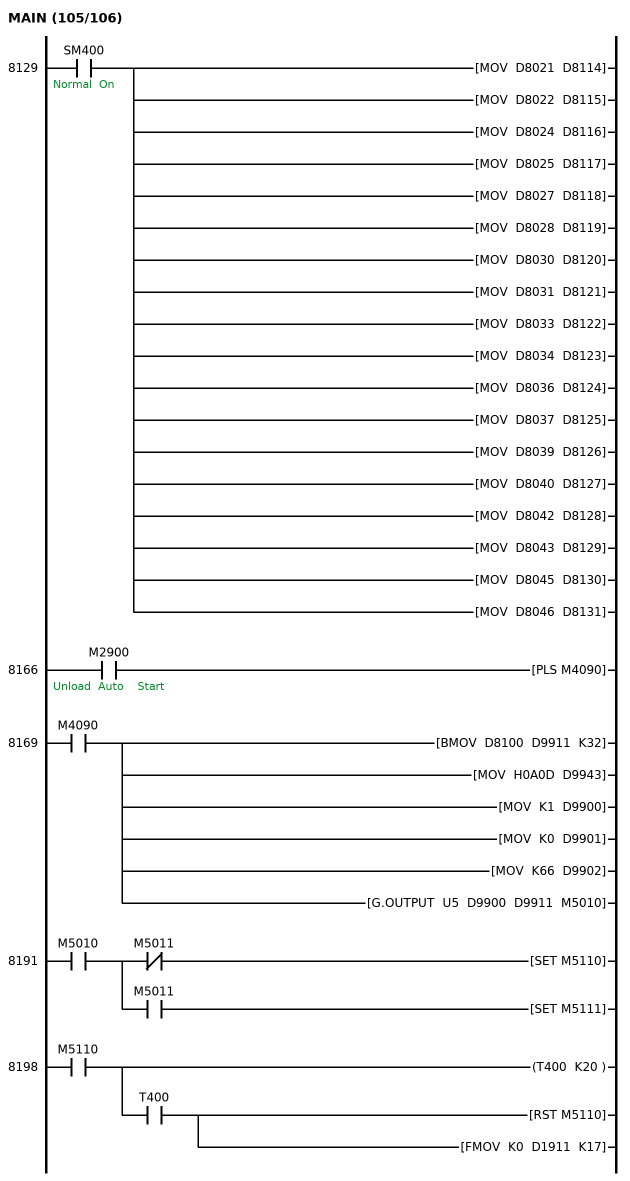
[picture p384: ladder of MAIN, rungs at steps 8129 to 8198]
8129  LD      SM400  ; Normal  On
      MOV     D8021 D8114
      MOV     D8022 D8115
      MOV     D8024 D8116
      MOV     D8025 D8117
      MOV     D8027 D8118
      MOV     D8028 D8119
      MOV     D8030 D8120
      MOV     D8031 D8121
      MOV     D8033 D8122
      MOV     D8034 D8123
      MOV     D8036 D8124
      MOV     D8037 D8125
      MOV     D8039 D8126
      MOV     D8040 D8127
      MOV     D8042 D8128
      MOV     D8043 D8129
      MOV     D8045 D8130
      MOV     D8046 D8131
8166  LD      M2900  ; Unload  Auto    Start
      PLS     M4090
8169  LD      M4090
      BMOV    D8100 D9911 K32
      MOV     H0A0D D9943
      MOV     K1 D9900
      MOV     K0 D9901
      MOV     K66 D9902
      G.OUTPUT U5 D9900 D9911 M5010
8191  LD      M5010
      MPS
      ANI     M5011
      SET     M5110
      MPP
      AND     M5011
      SET     M5111
8198  LD      M5110
      OUT     T400 K20
      AND     T400
      RST     M5110
      FMOV    K0 D1911 K17
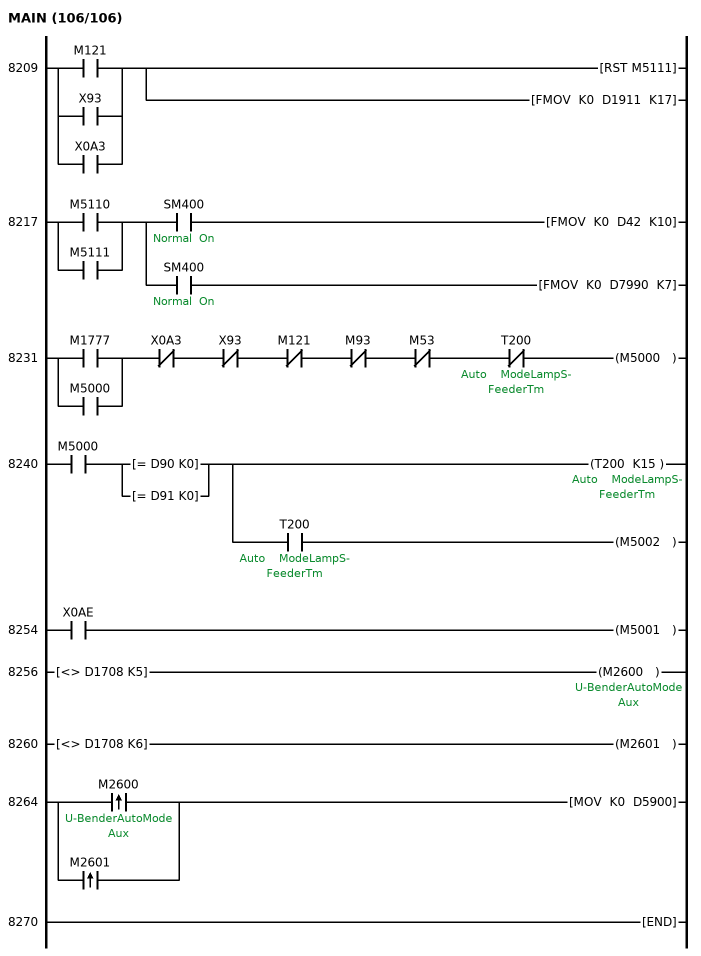
8209  LD      M121
      OR      X93
      OR      X0A3
      RST     M5111
      FMOV    K0 D1911 K17
8217  LD      M5110
      OR      M5111
      MPS
      AND     SM400  ; Normal  On
      FMOV    K0 D42 K10
      MPP
      AND     SM400  ; Normal  On
      FMOV    K0 D7990 K7
8231  LD      M1777
      OR      M5000
      ANI     X0A3
      ANI     X93
      ANI     M121
      ANI     M93
      ANI     M53
      ANI     T200  ; Auto    ModeLampS-FeederTm
      OUT     M5000
8240  LD      M5000
      LD=     D90 K0
      OR=     D91 K0
      ANB
      OUT     T200 K15  ; Auto    ModeLampS-FeederTm
      AND     T200  ; Auto    ModeLampS-FeederTm
      OUT     M5002
8254  LD      X0AE
      OUT     M5001
8256  LD<>    D1708 K5
      OUT     M2600  ; U-BenderAutoModeAux
8260  LD<>    D1708 K6
      OUT     M2601
8264  LDP     M2600  ; U-BenderAutoModeAux
      ORP     M2601
      MOV     K0 D5900
8270  END
END_PROGRAM

// device comments not shown above
D2  ; 150Ton  AutoBuff
R600  ; +OT Set PositionAxis-01
X31  ; f
X4B  ; Reset   #3
X4D  ; Reset   #2
X55  ; Carriage"B" OL
X56  ; Carriage"C" OL
X57  ; Carriage"D" OL
X58  ; Carriage"E" OL
X59  ; Carriage"F" OL
X80  ; NotchingSafety  Det'
X25D  ; NotchingR-SafetyDet'
X26B  ; NotchingR-Screp C/V OL
X303  ; 150Ton  BackPushUp Px
X304  ; 150Ton  BackPushDown Px
X305  ; 150Ton  SidePush1W-DetPx
X306  ; 150Ton  SidePush1RevPx
X30B  ; 150Ton  Safety#1Ls
X30C  ; 150Ton  Press UpPx
X30D  ; 150Ton  PressMidDet'Px
X30E  ; 150Ton  Press DnPx
X30F  ; 150Ton  PressureCheck
X313  ; 150Ton  Stopp UpPx
X314  ; 150Ton  Stopp DnPx
X315  ; 150Ton  SidePush2W-DetPx
X316  ; 150Ton  SidePush2Rev Px
X319  ; NotchingOil TempHigh
X31A  ; NotchingHi Press
X31B  ; 150Ton  Safety#1Ls
X31C  ; 150Ton  Side    L-Safety
X31D  ; 150Ton  Side    R-Safety
X31E  ; 150Ton  Hyd'TankTempHigh
X31F  ; 150Ton  Hyd'TankTempLow
X487  ; Buffer  Work    Stop
X490  ; Divert#2WorkDet'#1
X49E  ; Z-BenderHyd' OilTemp Hi
X54C  ; L-BendOtSideMoldPOt Fwd
X54D  ; L-BendOtSideMoldPOt Rev
X5CC  ; U-BendOtSideMoldPin Fwd
X5CD  ; U-BendOtSideMoldPin Rev
X5CE  ; U-BendOtUp GuideFwd
X600  ; U-BendInConv' Up
X601  ; U-BendInConv' Dn
X660  ; U-BendOtConv' Up
X661  ; U-BendOtConv' Dn
X6C0  ; Unload  Transfer+ OT
X6C1  ; Unload  TransferHome
X6C2  ; Unload  Transfer- OT
X6C8  ; Unload  TransferUp
X6C9  ; Unload  TransferDown
X6CA  ; Unload  Head    Clamp Px
X6CB  ; Unload  Head    Unclamp Px
X720  ; NEW SHEARING DIV. DN
X762  ; Buffer  Conv' OL
Y0B9  ; Buffer  Conv'Mc
Y0E4  ; Cycle Time Hold
Y0E5  ; Cycle Time Reset
Y1B6  ; Lifter  Up/Down Slow
Y1B7  ; Lifter  Up/Down Reset
Y2AA  ; NotchingRellief Sv
Y320  ; 150Ton  BackPushUp Sv
Y321  ; 150Ton  BackPushDn Sv
Y324  ; 150Ton  SidePushFwd Sv
Y325  ; 150Ton  SidePushRev Sv
Y326  ; NotchingHi PressSv
Y328  ; 150Ton  Stopper Up Sv
Y329  ; 150Ton  Stopper Dn Sv
Y32B  ; 150Ton  Press UpSv
Y32C  ; 150Ton  Press DnSv
Y32D  ; 150Ton  Rellief Sv
Y32E  ; 150Ton  Exhaust Sv
Y32F  ; 150Ton  WheelingSv
Y414  ; L-BenderRellief Sv
Y4AB  ; Z-BednerUp Sv
Y634  ; U-BendInSideGuidFwd Sv
Y694  ; U-BendOtSideGuidFwd Sv
Y6E0  ; Unload  TransferUp Sv
Y6E1  ; Unload  TransferDn Sv
Y74D  ; OutConv'#44MotorMc
Y74E  ; OutConv'#45MotorMc
Y79C  ; m43 cv lift up sol
M243  ; Divert#2On At
M248  ; Taping#1Work    Finish  Set
M278  ; IdleConvWork    Finish  Set
M282  ; IdleConvOn At
M283  ; U-BenderServo GoAt
M284  ; U-BenderOn At
M285  ; U-BenderOff At
M1001  ; Carriage"A" Set Sw
M1002  ; Carriage"B" Set Sw
M1003  ; Carriage"C" Set Sw
M1004  ; Carriage"D" Set Sw
M1005  ; Carriage"E" Set Sw
M1014  ; Sheet   Feeder  "E" Pos'Set Sw
M1015  ; Sheet   Feeder  "F" Pos'Set Sw
M1016  ; Sheet   Feeder  ConvPos'Set Sw
M1020  ; Sheet   Feeder  "A" Pos'Set Lp
M1021  ; Sheet   Feeder  "B" Pos'Set Lp
M1022  ; Sheet   Feeder  "C" Pos'Set Lp
M1023  ; Sheet   Feeder  "D" Pos'Set Lp
M1024  ; Sheet   Feeder  "E" Pos'Set Lp
M1025  ; Sheet   Feeder  "F" Pos'Set Lp
M1026  ; Sheet   Feeder  ConvPos'Set Lp
M1079  ; Carriage#2 Pos'  Fault
M1081  ; Carriage#4 Pos'  Fault
M1082  ; Carriage#5 Pos'  Fault
M1083  ; Carriage#6 Pos'  Fault
M1090  ; CarriagePositionOK
M1098  ; S/F     CarriageOK
M1102  ; S/F     Working Order Ok
M1118  ; S/F Car'PositionGo Aux.
M1230  ; 2-Axis  PositionOK
M1231  ; 3-Axis  PositionOK
M1232  ; 4-Axis  PositionOK
M1233  ; 5-Axis  PositionOK
M1234  ; 6-Axis  PositionOK
M1235  ; 7-Axis  PositionOK
M1236  ; 8-Axis  PositionOK
M1237  ; 2-Axis  PositionOK
M1238  ; 16-Axis PositionOK
M1316  ; NotchingMidStoppDown At
M1333  ; NotchingMid SidePush    Fwd At
M1401  ; 150Ton  Auto    Mode
M1402  ; 150Ton  Manual  Mode
M1410  ; 150Ton  Hold Sw
M1420  ; 150Ton  Press   Pass    Model
M1425  ; 150Ton  Working Model   Detect
M1430  ; 12-Axis PositionOK
M1431  ; 13-Axis PositionOK
M1439  ; 150Ton  All-AxisPos' OK
M1452  ; 150Ton  Press   Up Hm
M1453  ; 150Ton  BackPushRev Hm
M1454  ; 150Ton  BackPushDown Hm
M1455  ; 150Ton  Stopper Down Hm
M1456  ; 150Ton  SidePushRev Hm
M1471  ; 150Ton  Conv'RunEnable
M1472  ; 150Ton  ServoRunEnable
M1520  ; 150Ton  Press   Up Hm At
M1521  ; 150Ton  Stopper Up At
M1522  ; 150Ton  BackPushRev At
M1523  ; 150Ton  BackPushUp At
M1524  ; 150Ton  BackPushFwd At
M1525  ; 150Ton  SidePushFwd At
M1526  ; 150Ton  SidePush34Fwd At
M1528  ; 150Ton  Press   Down At
M1533  ; 150Ton  Press   Up At
M1534  ; 150Ton  SidePushBwd At
M1535  ; 150Ton  BackPushBwd At
M1536  ; 150Ton  SidePush#34BwdAt
M1537  ; 150Ton  BackPushDown At
M1538  ; 150Ton  Stopper Down At
M1560  ; 150Ton  Press   Stop
M1580  ; 150Ton  AutoStep0
M1581  ; 150Ton  AutoStep1
M1582  ; 150Ton  AutoStep2
M1583  ; 150Ton  AutoStep3
M1584  ; 150Ton  AutoStep4
M1585  ; 150Ton  AutoStep5
M1586  ; 150Ton  AutoStep6
M1720  ; 150Ton  ConveyorOn At
M1721  ; TurnoverInConv' On At
M1722  ; 150Ton=>TurnoverIn Move Ok
M1724  ; TurnoverInConv' On At
M1735  ; TurnoverOutCent'Bwd At
M1738  ; TurnoverIn Retn At
M1740  ; Turn In Center' Fwd At
M1741  ; Turn In Center' Ok
M1742  ; Turn In Center' Rev At
M1770  ; Turn In ConvSlowSet
M1781  ; TurnoverAutoStep1
M1782  ; TurnoverAutoStep2
M1930  ; Turn OutCenter' Set
M2120  ; Center#1Fwd At
M2122  ; Center#3Fwd At
M2130  ; Center  Ok
M2132  ; Center#1Rev At
M2133  ; Center#3Rev At
M2151  ; Divert#3OutConv'SlowAt
M2181  ; Divert#2AutoStep1
M2182  ; Divert#2AutoStep2
M2183  ; Divert#2AutoStep3
M2184  ; Divert#2AutoStep4
M2311  ; L-BenderClamp AtFrontMdl
M2312  ; L-BenderClamp AtRear Mdl
M2315  ; L-BenderOtPush#2Fwd At
M2316  ; L-BenderInPush#1Fwd At
M2317  ; L-BenderOtPush#1Fwd At
M2744  ; Guide   Rev At
M2758  ; Upper   Knife   Turn Ok
M2936  ; Head    Unclamp At
M2973  ; Rev Slow
M2987  ; Unload  AutoStep7
M3146  ; OutConv'#35DivetUp At
M3157  ; OutConv'#37DivetUp At
M3158  ; OutConv'#37DivetDn At
M3159  ; OutConv'#35DivetUp At
M3176  ; OutConv'#37DivetUp At
M3178  ; OutConv'#37DivetDn At
M3312  ; OutConv'#43MotorMn On
M3313  ; OutConv'#44MotorMn On
M3321  ; OutConv'#32MotorPass Off
M3322  ; OutConv'#33MotorPass Off
M3323  ; OutConv'#34MotorPass Off
M3324  ; OutConv'#35MotorPass Off
M3325  ; OutConv'#36MotorPass Off
M3326  ; OutConv'#37MotorPass Off
M3327  ; OutConv'#38MotorPass Off
M3328  ; OutConv'#39MotorPass Off
M3329  ; OutConv'#40MotorPass Off
M3330  ; OutConv'#41MotorPass Off
M3331  ; OutConv'#42MotorPass Off
M3332  ; OutConv'#43MotorPass Off
M3333  ; OutConv'#44MotorPass Off
M3401  ; L-BenderWork    Model Ok
M3421  ; L-BendInMoldChanAutoStep1
M3422  ; L-BendInMoldChanAutoStep2
M3423  ; L-BendInMoldChanAutoStep3
M3424  ; L-BendInMoldChanAutoStep4
M3425  ; L-BendInMoldChanAutoStep5
M3426  ; L-BendInMoldChanAutoStep6
M3427  ; L-BendInMoldChanAutoStep7
M3428  ; Ready   Pos'+ >-Mode Set
M3429  ; Ready   Pos'- >+Mode Set
M3434  ; L-BendInSideMoldPin Rev At
M3436  ; Mold PinFwd At
M3444  ; L-BendInNow MoldGo
M3445  ; 7.Axis  PosStartOk
M3446  ; 7.Axis  Pos' Ok
M3447  ; L-BendInSideMoldPin Rev At
M3449  ; L-BendInNow PushMold Go
M3453  ; Pos Ok
M3454  ; 7.Axis  Pos' Ok
M3455  ; Mold    Clamp At
M3461  ; L-BendOtMoldChanAutoStep1
M3462  ; L-BendOtMoldChanAutoStep2
M3463  ; L-BendOtMoldChanAutoStep3
M3464  ; L-BendOtMoldChanAutoStep4
M3465  ; L-BendOtMoldChanAutoStep5
M3466  ; L-BendOtMoldChanAutoStep6
M3467  ; L-BendOtMoldChanAutoStep7
M3468  ; Ready   Pos'   +Mode Set
M3469  ; Ready   Pos'   -Mode Set
M3474  ; L-BendOtSideMoldPin Rev At
M3476  ; Mold PinFwd At
M3484  ; L-BendOtNow MoldGo
M3485  ; 8.Axis  PosStartOk
M3486  ; 8.Axis  Pos' Ok
M3487  ; L-BendOtSideMoldPin Rev At
M3492  ; PositionOk
M3501  ; U-BenderWork    Model Ok
M3502  ; U-BendOtMoldDataPos'Ok
M3520  ; U-BendInMoldChanAutoStep0
M3521  ; U-BendInMoldChanAutoStep1
M3522  ; U-BendInMoldChanAutoStep2
M3523  ; U-BendInMoldChanAutoStep3
M3524  ; U-BendInMoldChanAutoStep4
M3525  ; U-BendInMoldChanAutoStep5
M3526  ; U-BendInMoldChanAutoStep6
M3527  ; U-BendInMoldChanAutoStep7
M3528  ; Ready   Pos'- >+Mode Set
M3529  ; Ready   Pos'+ >-Mode Set
M3534  ; U-BendInSideMoldPin Rev At
M3536  ; U-BendInSideMoldPin Fwd At
M3544  ; U-BendInNow MoldGo
M3545  ; 12.Axis Pos' Ok
M3546  ; 12.Axis  Pos' Ok
M3547  ; U-BendInSideMoldPin Rev At
M3560  ; U-BendOtMoldChanAutoStep0
M3561  ; U-BendOtMoldChanAutoStep1
M3562  ; U-BendOtMoldChanAutoStep2
M3563  ; U-BendOtMoldChanAutoStep3
M3564  ; U-BendOtMoldChanAutoStep4
M3565  ; U-BendOtMoldChanAutoStep5
M3566  ; U-BendOtMoldChanAutoStep6
M3567  ; U-BendOtMoldChanAutoStep7
M3568  ; Ready   Pos'   +Mode Set
M3569  ; Ready   Pos'   -Mode Set
M3574  ; U-BendOtSideMoldPin Rev At
M3576  ; U-BendOtSideMoldPin Fwd At
M3584  ; U-BendOtNow MoldGo
M3585  ; 13.Axis PosStartOk
M3586  ; 13.Axis  Pos' Ok
M3587  ; U-BendOtSideMoldPin Rev At
M3588  ; U-BendOtMold    Unclamp At
M3594  ; 13.Axis PosStartOk
M4135  ; System  Error   Reset   Axis-01
M4136  ; Servo   Error   Reset   Axis-01
M4155  ; System  Error   Reset   Axis-02
M4156  ; Servo   Error   Reset   Axis-02
M4175  ; System  Error   Reset   Axis-03
M4176  ; Servo   Error   Reset   Axis-03
M4195  ; System  Error   Reset   Axis-04
M4196  ; Servo   Error   Reset   Axis-04
M4215  ; System  Error   Reset   Axis-05
M4216  ; Servo   Error   Reset   Axis-05
M4235  ; System  Error   Reset   Axis-06
M4236  ; Servo   Error   Reset   Axis-06
M4255  ; System  Error   Reset   Axis-07
M4256  ; Servo   Error   Reset   Axis-07
M4275  ; System  Error   Reset   Axis-08
M4276  ; Servo   Error   Reset   Axis-08
M4295  ; System  Error   Reset   Axis-09
M4296  ; Servo   Error   Reset   Axis-09
M4315  ; System  Error   Reset   Axis-10
M4316  ; Servo   Error   Reset   Axis-10
M4335  ; System  Error   Reset   Axis-11
M4336  ; Servo   Error   Reset   Axis-11
M4355  ; System  Error   Reset   Axis-12
M4356  ; Servo   Error   Reset   Axis-12
M4375  ; System  Error   Reset   Axis-13
M4376  ; Servo   Error   Reset   Axis-13
M4388  ; Servo   Stop    Axis-14
M4390  ; JOG +   Axis-14
M4391  ; JOG -   Axis-14
M4395  ; System  Error   Reset   Axis-14
M4396  ; Servo   Error   Reset   Axis-14
M4415  ; System  Error   Reset   Axis-15
M4416  ; Servo   Error   Reset   Axis-15
M4428  ; Servo   Stop    Axis-16
M4430  ; JOG +   Axis-16
M4431  ; JOG -   Axis-16
M4435  ; System  Error   Reset   Axis-16
M4436  ; Servo   Error   Reset   Axis-16
M4455  ; System  Error   Reset   Axis-17
M4456  ; Servo   Error   Reset   Axis-17
M4475  ; System  Error   Reset   Axis-18
M4476  ; Servo   Error   Reset   Axis-18
M4495  ; System  Error   Reset   Axis-19
M4496  ; Servo   Error   Reset   Axis-19
M4515  ; System  Error   Reset   Axis-20
M4516  ; Servo   Error   Reset   Axis-20
M4535  ; System  Error   Reset   Axis-21
M4536  ; Servo   Error   Reset   Axis-21
M4555  ; System  Error   Reset   Axis-22
M4556  ; Servo   Error   Reset   Axis-22
M4575  ; System  Error   Reset   Axis-23
M4576  ; Servo   Error   Reset   Axis-23
M4595  ; System  Error   Reset   Axis-24
M4596  ; Servo   Error   Reset   Axis-24
M4615  ; System  Error   Reset   Axis-25
M4616  ; Servo   Error   Reset   Axis-25
M4635  ; System  Error   Reset   Axis-26
M4636  ; Servo   Error   Reset   Axis-26
M4655  ; System  Error   Reset   Axis-27
M4656  ; Servo   Error   Reset   Axis-27
M4675  ; System  Error   Reset   Axis-28
M4676  ; Servo   Error   Reset   Axis-28
M4695  ; System  Error   Reset   Axis-29
M4696  ; Servo   Error   Reset   Axis-29
M4715  ; System  Error   Reset   Axis-30
M4716  ; Servo   Error   Reset   Axis-30
M4728  ; Servo   Stop    Axis-31
M4730  ; JOG +   Axis-30
M4731  ; JOG -   Axis-30
M4770  ; 2.Axis  Busy
M4771  ; 3.Axis  Busy
M4772  ; 4.Axis  Busy
M4773  ; 5.Axis  Busy
M4774  ; 6.Axis  Busy
M4775  ; 7.Axis  Busy
M4776  ; 8.Axis  Busy
M4777  ; 9.Axis  Busy
M4778  ; 10.Axis  Busy
M4779  ; 11.Axis  Busy
M4780  ; 12.Axis  Busy
M4782  ; 14.Axis  Busy
M4784  ; 16.Axis  Busy
M4785  ; 17.Axis  Busy
M4786  ; 18.Axis  Busy
M4787  ; 19.Axis  Busy
M4789  ; 21.Axis  Busy
M4791  ; 23.Axis  Busy
M4799  ; 31.Axis  Busy
M4800  ; 32.Axis  Busy
M5395  ; System  Error   Axis-12
M5396  ; Servo   Error   Axis-12
M5443  ; Servo   Ready   Axis-14
M5475  ; System  Error   Axis-16
M5476  ; Servo   Error   Axis-16
M5483  ; Servo   Ready   Axis-16
M5783  ; 31.Axis Servo   Ready
M6083  ; NotchingSidePush#2FwdFlt
M6084  ; NotchingSidePush#2BwdFlt
M6107  ; #7 ~ #8 Safety  ClashFlt
M7260  ; Unload  TransferOL Fault
M7313  ; 14.Axis OverRun Fault
M7315  ; 16.Axis OverRun Fault
M7330  ; 31.Axis OverRun Fault
M7331  ; 32.Axis OverRun Fault
L2  ; 150 Ton Working Latch
L13  ; 150Ton->TurnoverLatch
L55  ; Taping->Taping#2Work    Latch
L59  ; Divert#2Work    Latch
L60  ; Divert#2=>L-bendLetch
L61  ; Carriage"A" Set Lp
L62  ; Carriage"B" Set Lp
L63  ; Carriage"C" Set Lp
L64  ; Carriage"D" Set Lp
L65  ; Carriage"E" Set Lp
L81  ; #32->M33Work    Latch
L91  ; #42->M43Work    Latch
L92  ; #43->M44Work    Latch
L93  ; #44->M45Work    Latch
L95  ; #36MotorWorkStopLatch
B0D  ; 14.Axis Set     PositionOk
B1E  ; 31.Axis Set     PositionOk
B1F  ; 32.Axis Set     PositionOk
B20  ; 01.Axis Ready   PositionOk
B21  ; 02.Axis Ready   PositionOk
B22  ; 03.Axis Ready   PositionOk
B23  ; 04.Axis Ready   PositionOk
B24  ; 05.Axis Ready   PositionOk
B25  ; 06.Axis Ready   PositionOk
B26  ; 07.Axis Ready   PositionOk
B27  ; 08.Axis Ready   PositionOk
B28  ; 09.Axis Ready   PositionOk
B29  ; 10.Axis Ready   PositionOk
B2A  ; 11.Axis Ready   PositionOk
B2B  ; 12.Axis Ready   PositionOk
B2D  ; 14.Axis Ready   PositionOk
B2F  ; 16.Axis Ready   PositionOk
B30  ; 17.Axis Ready   PositionOk
B31  ; 18.Axis Ready   PositionOk
B32  ; 19.Axis Ready   PositionOk
B34  ; 21.Axis Ready   PositionOk
B3E  ; 31.Axis Ready   PositionOk
B3F  ; 32.Axis Ready   PositionOk
B41  ; NotchingPress #2Use Set
B42  ; NotchingPress #3Use Set
B43  ; NotchingPress #4Use Set
B44  ; NotchingPress #5Use Set
B45  ; NotchingPress #6Use Set
B46  ; NotchingPress #7Use Set
B47  ; NotchingPress #8Use Set
B4C  ; NotchingPress #9UseSw
B4D  ; NotchingPress#10UseSw
B50  ; 150Ton  PressUseSet
B5C  ; 29.Axis Middle  PositionOk
B83  ; S/F     Conv'
B87  ; NotchingConv'
B8B  ; 150Ton  Conv'
B8F  ; Turn In Conv'
B93  ; Turn OutConv'
B97  ; Roll    Conv'
B9B  ; Divert#1In Conv'
B9F  ; Divert#2In Conv'
B0C3  ; Z-BenderHyd'PumpOn Sw
B10A  ; Cycle TmAllResetSw
B110  ; JogSpeedFast #2
B111  ; Pitch   Mode #2
B112  ; Edit    Mode#2
B113  ; Pitch   Mode #2 L-Bender
B11F  ; Press   Working Set Lp
B140  ; S/F HeadUpSw
B141  ; S/F HeadDownSw
B142  ; S/F HeadVacuum  OnSw
B143  ; S/F HeadVacuum  OffSw
B160  ; Sheet#1 Set Sw
B170  ; Jog FastSpeed SwS-Feeder
B171  ; Jog     /MDI Sw S-Feeder
B1D1  ; Lifter  DnSw
B24E  ; MICON ON
B250  ; Carriage"C" Fwd Sw
B251  ; Carriage"C" Rev Sw
B252  ; Carriage"C"Roll Fwd Sw
B253  ; Carriage"C"Roll Rev Sw
B25C  ; S/F HeadVacuum  OnSw
B25D  ; S/F HeadVacuum  OffSw
B25E  ; S/F HeadVacuum  On #3 Sw
B25F  ; S/F HeadVacuum  #3 OffSw
B260  ; S/F HeadVacuum  On #4 Sw
B261  ; S/F HeadVacuum  #4 OffSw
B264  ; S/F ConvCenteri'Fwd #2  Sw
B265  ; S/F ConvCenteri'Rev #2  Sw
B266  ; S/F ConvCenteri'Fwd #3  Sw
B267  ; S/F ConvCenteri'Rev #3  Sw
B2A9  ; L-BenderJog HighSpeed Sw
B2AB  ; U-BenderJog HighSpeed Sw
B320  ; 150Ton  BackPushUp Sw
B321  ; 150Ton  BackPushDn Sw
B324  ; 150Ton  SidePushFwd Sw
B325  ; 150Ton  SidePushRev Sw
B328  ; 150Ton  Stopper Up Sw
B329  ; 150Ton  Stopper Dn Sw
B32B  ; 150Ton  Press UpSw
B32C  ; 150Ton  Press DnSw
B32D  ; 150Ton  Rellief Sw
B32E  ; 150Ton  Exhaust Sw
B32F  ; 150Ton  WheelingSw
B3AA  ; Roll    AirBlow Off Sw
B4A7  ; Divert#2Center' Rev Aux.
B4AB  ; Z-BednerUp Sw
B500  ; L-Bend  Conv' UpSw Aux
B510  ; L-Bend  Conv' UpSw Lp
B52B  ; L-BenderRellief Sw
B52C  ; L-BendInMold PinFwd Sw
B52D  ; L-BendInMold PinRev Sw
B56C  ; L-BendOtMold PinFwd Sw
B56D  ; L-BendOtMold PinRev Sw
B588  ; Z-bend  Clamp UpSw
B598  ; Z-bend  Clamp UpSw Lp
B5E2  ; U-BendOtSide CmpUnit FwdSw
B5E3  ; U-BendOtSide CmpUnit RevSw
B600  ; U-Bend  Conv' UpSw
B610  ; U-Bend  Conv' UpLp
B630  ; U-BendInSideMoldPin Fwd Sw
B631  ; U-BendInSideMoldPin Rev Sw
B632  ; U-BendInSideMoldPinClampSw
B633  ; U-BendInSideMoldPinUncmpSw
B634  ; U-BendInSideGuidFwd Sw
B660  ; U-BendInUp GuideFwd Sw
B670  ; U-Bend  SideMoldPin Fwd Sw Lp
B690  ; U-BendOtSideMoldPin Fwd Sw
B691  ; U-BendOtSideMoldPin Rev Sw
B692  ; U-BendOtSideMoldPinClampSw
B693  ; U-BendOtSideMoldPinUncmpSw
B694  ; U-BendOtSideGuidFwd Sw
B69E  ; U-BendOtStopper Rev Sw
B6E0  ; Unload  TransferUp Sw
B6E1  ; Unload  TransferDn Sw
B6E2  ; Unload  TransferHead    Clamp Sw
B6E3  ; Unload  TransferHead    Uncmp Sw
B750  ; Lifter  UpSw
B751  ; Lifter  DnSw
B0AA3  ; Divert#2Ot Conv'
B0AAB  ; Idle    Conv'
B0AAF  ; U-BenderConv'
B0E34  ; Home    ReturnSwIdle
B0E35  ; Home    ReturnLpIdle
B0E54  ; Home    ReturnSwRoller
B0E55  ; Home    ReturnLpRoller
B0F2E  ; Z-BenderWork    Notuser Lp
B0F34  ; Home    ReturnSwTaping
B0F35  ; Home    ReturnLpTaping
B100D  ; +OT     Fault   Axis-14
B100F  ; +OT     Fault   Axis-16
B101E  ; +OT     Fault   Axis-31
B101F  ; +OT     Fault   Axis-32
B102D  ; -OT     Fault   Axis-14
B102F  ; -OT     Fault   Axis-16
B103E  ; -OT     Fault   Axis-31
B103F  ; -OT     Fault   Axis-32
B108D  ; Jog Set Axis-14
B108F  ; Jog Set Axis-16
B109E  ; 31.Axis Jog Set
B109F  ; 32.Axis Jog Set
B10C1  ; 02.Axis HmReturnSet
B10C2  ; 03.Axis HmReturnSet
B10C3  ; 04.Axis HmReturnSet
B10C4  ; 05.Axis HmReturnSet
B10C5  ; 06.Axis HmReturnSet
B10C6  ; 07.Axis HmReturnSet
B10C7  ; 08.Axis HmReturnSet
B10C8  ; 09.Axis HmReturnSet
B10C9  ; 10.Axis HmReturnSet
B10CA  ; 11.Axis HmReturnSet
B10CB  ; 12.Axis HmReturnSet
B10CC  ; 13.Axis HmReturnSet
B10CD  ; 14.Axis HmReturnSet
B10CE  ; 15.Axis HmReturnSet
B10CF  ; 16.Axis HmReturnSet
B10D0  ; 17.Axis HmReturnSet
B10D1  ; 18.Axis HmReturnSet
B10D2  ; 19.Axis HmReturnSet
B10D3  ; 20.Axis HmReturnSet
B10D4  ; 21.Axis HmReturnSet
B10D5  ; 22.Axis HmReturnSet
B10D6  ; 23.Axis HmReturnSet
B10D7  ; 24.Axis HmReturnSet
B10D8  ; 25.Axis HmReturnSet
B10D9  ; 26.Axis HmReturnSet
B10DA  ; 27.Axis HmReturnSet
B10DB  ; 28.Axis HmReturnSet
B10DC  ; 29.Axis HmReturnSet
B10DD  ; 30.Axis HmReturnSet
B10DE  ; 31.Axis HmReturnSet
B10DF  ; 32.Axis HmReturnSet
B10E0  ; S/FTransModelNo.Ok
B10E1  ; Center' ModelNo.Ok
B10E3  ; 150Ton  ModelNo.Ok
B10E4  ; Turn In ModelNo.Ok
B10E5  ; Turn Ot ModelNo.Ok
B10F0  ; Divert#1ModelNo.Ok
B10F1  ; Buffer  ModelNo.Ok
B10F2  ; Divert#2ModelNo.Ok
B10F4  ; IdleConvModelNo.Ok
B1101  ; 02.Axis Data SetReady
B1102  ; 03.Axis Data SetReady
B1103  ; 04.Axis Data SetReady
B1104  ; 05.Axis Data SetReady
B1105  ; 06.Axis Data SetReady
B1106  ; 07.Axis Data SetReady
B1107  ; 08.Axis Data SetReady
B110D  ; 14.Axis Data SetReady
B110E  ; 15.Axis Data SetReady
B110F  ; 16.Axis Data SetReady
B1113  ; 20.Axis Data SetReady
B1114  ; 21.Axis Data SetReady
B1115  ; 22.Axis Data SetReady
B1116  ; 23.Axis Data SetReady
B1117  ; 24.Axis Data SetReady
B1118  ; 25.Axis Data SetReady
B1119  ; 26.Axis Data SetReady
B111B  ; 28.Axis Data SetReady
B111C  ; 29.Axis Data SetReady
B111D  ; 30.Axis Data SetReady
B111E  ; 31.Axis Data SetReady
B111F  ; 32.Axis Data SetReady
B1120  ; 01.Axis Data SetSw
B1121  ; 02.Axis Data SetSw
B1122  ; 03.Axis Data SetSw
B1123  ; 04.Axis Data SetSw
B1124  ; 05.Axis Data SetSw
B1125  ; 06.Axis Data SetSw
B1126  ; 07.Axis Data SetSw
B1127  ; 08.Axis Data SetSw
B1128  ; 09.Axis Data SetSw
B1129  ; 10.Axis Data SetSw
B112A  ; 11.Axis Data SetSw
B112B  ; 12.Axis Data SetSw
B112C  ; 13.Axis Data SetSw
B112D  ; 14.Axis Data SetSw
B112E  ; 15.Axis Data SetSw
B112F  ; 16.Axis Data SetSw
B1130  ; 17.Axis Data SetSw
B1131  ; 18.Axis Data SetSw
B1132  ; 19.Axis Data SetSw
B1133  ; 20.Axis Data SetSw
B1134  ; 21.Axis Data SetSw
B1135  ; 22.Axis Data SetSw
B1136  ; 23.Axis Data SetSw
B1137  ; 24.Axis Data SetSw
B1138  ; 25.Axis Data SetSw
B1139  ; 26.Axis Data SetSw
B113A  ; 27.Axis Data SetSw
B113B  ; 28.Axis Data SetSw
B113C  ; 29.Axis Data SetSw
B113D  ; 30.Axis Data SetSw
B113E  ; 31.Axis Data SetSw
B113F  ; 32.Axis Data SetSw
B1140  ; 01.Axis Data SetLp
B1141  ; 02.Axis Data SetLp
B1142  ; 03.Axis Data SetLp
B1143  ; 04.Axis Data SetLp
B1144  ; 05.Axis Data SetLp
B1145  ; 06.Axis Data SetLp
B1146  ; 07.Axis Data SetLp
B1147  ; 08.Axis Data SetLp
B1148  ; 09.Axis Data SetLp
B1149  ; 10.Axis Data SetLp
B114A  ; 11.Axis Data SetLp
B114B  ; 12.Axis Data SetLp
B114C  ; 13.Axis Data SetLp
B114D  ; 14.Axis Data SetLp
B114E  ; 15.Axis Data SetLp
B114F  ; 16.Axis Data SetLp
B1150  ; 17.Axis Data SetLp
B1151  ; 18.Axis Data SetLp
B1152  ; 19.Axis Data SetLp
B1153  ; 20.Axis Data SetLp
B1154  ; 21.Axis Data SetLp
B1155  ; 22.Axis Data SetLp
B1156  ; 23.Axis Data SetLp
B1157  ; 24.Axis Data SetLp
B1158  ; 25.Axis Data SetLp
B1159  ; 26.Axis Data SetLp
B115A  ; 27.Axis Data SetLp
B115B  ; 28.Axis Data SetLp
B115C  ; 29.Axis Data SetLp
B115D  ; 30.Axis Data SetLp
B115E  ; 31.Axis Data SetLp
B115F  ; 32.Axis Data SetLp
B116D  ; 14.Axis PositionStart
B116F  ; 16.Axis PositionStart
B117E  ; 31.Axis PositionStart
B117F  ; 32.Axis PositionStart
B118D  ; 14.Axis  Busy
B118F  ; 16.Axis  Busy
B119E  ; 31.Axis  Busy
B119F  ; 32.Axis  Busy
B11AD  ; 14.Axis Stop
B11AF  ; 16.Axis Stop
B11BE  ; 31.Axis Stop
B11BF  ; 32.Axis Stop
B11C0  ; 01.Axis FwdPitchSw
B11C2  ; 03.Axis FwdPitchSw
B11C3  ; 04.Axis FwdPitchSw
B11C4  ; 05.Axis FwdPitchSw
B11C5  ; 06.Axis FwdPitchSw
B11C6  ; 07.Axis FwdPitchSw
B11C7  ; 08.Axis FwdPitchSw
B11C8  ; 09.Axis FwdPitchSw
B11C9  ; 10.Axis FwdPitchSw
B11CA  ; 11.Axis FwdPitchSw
B11CD  ; 14.Axis FwdPitchSw
B11CE  ; 15.Axis FwdPitchSw
B11CF  ; 16.Axis FwdPitchSw
B11D0  ; 17.Axis FwdPitchSw
B11D4  ; 21.Axis FwdPitchSw
B11D5  ; 22.Axis FwdPitchSw
B11D6  ; 23.Axis FwdPitchSw
B11D7  ; 24.Axis FwdPitchSw
B11DD  ; 30.Axis FwdPitchSw
B11DE  ; 31.Axis FwdPitchSw
B11DF  ; 32.Axis FwdPitchSw
B11E0  ; 01.Axis RevPitchSw
B11E1  ; 02.Axis RevPitchSw
B11E2  ; 03.Axis RevPitchSw
B11E3  ; 04.Axis RevPitchSw
B11E4  ; 05.Axis RevPitchSw
B11E5  ; 06.Axis RevPitchSw
B11E6  ; 07.Axis RevPitchSw
B11E7  ; 08.Axis RevPitchSw
B11E8  ; 09.Axis RevPitchSw
B11E9  ; 10.Axis RevPitchSw
B11EA  ; 11.Axis RevPitchSw
B11EC  ; 13.Axis RevPitchSw
B11ED  ; 14.Axis RevPitchSw
B11EE  ; 15.Axis RevPitchSw
B11EF  ; 16.Axis RevPitchSw
B11F0  ; 17.Axis RevPitchSw
B11F1  ; 18.Axis RevPitchSw
B11F2  ; 19.Axis RevPitchSw
B11F4  ; 21.Axis RevPitchSw
B11F5  ; 22.Axis RevPitchSw
B11F6  ; 23.Axis RevPitchSw
B11F7  ; 24.Axis RevPitchSw
B11FD  ; 30.Axis RevPitchSw
B11FE  ; 31.Axis RevPitchSw
B11FF  ; 32.Axis RevPitchSw
B14AB  ; Z-BednerDn Sw
T333  ; NotchingMid SidePush    ClampOK
T334  ; NotchingMidStoppUp OK
T335  ; NotchingMidStoppDn OK
T410  ; 150Ton  Press   Up OK
T412  ; 150Ton  BackPushFwd OK
T413  ; 150Ton  BackPushRev OK
T414  ; 150Ton  BackPushUp OK
T415  ; 150Ton  BackPushDown OK
T416  ; 150Ton  Stopper Up OK
T417  ; 150Ton  Stopper Down OK
T418  ; 150Ton  SidePushClamp OK
T419  ; 150Ton  SidePushRev OK
T420  ; 150Ton  Work    Empty
T421  ; 150Ton  SidePush#34FwdOK
T422  ; 150Ton  SidePush#34BwdOK
T424  ; 150Ton  Work    Ok Tm
T483  ; 150Ton  Hi-PressChk OK
T490  ; 150Ton  Hyd'PumpHeaterOn
T491  ; 150Ton  Hyd'PumpHeatOff
T494  ; 150Ton  Hyd'PumpOff Tm
T605  ; Buffer  Work    Entry Tm
T607  ; Buffer  Work    Stop Tm
T615  ; Divert#2Center' Fwd  Tm
T619  ; Divert#2Center' #1 Fwd  Tm
T621  ; Divert#2Center' #1 Rev  Tm
T622  ; Divert#2Center' #2 Fwd  Tm
T623  ; Divert#2Center' #2 Rev  Tm
T624  ; Divert#2Center' #3 Fwd  Tm
T625  ; Divert#2Center' #3 Rev  Tm
T690  ; 150Ton  Hyd'PumpOn Tm
T734  ; L-BendInPushUnitFwd Tm
T744  ; L-BendOtPushUnitFwd Tm
T1020  ; Lifter  WorkDet'Ok Tm
T1053  ; Divert#3OutConv'Run Tm
T1139  ; OutConv'#41 WorkStop Ph
T1156  ; M32->M33Auto RunTm
T1166  ; M42->M43Auto RunTm
T1167  ; M43->M44Auto RunTm
T1168  ; M44->M45Auto RunTm
T1171  ; M32->M33Auto RunOver Tm
T1181  ; M42->M43Auto RunOver Tm
T1182  ; M43->M44Auto RunOver Tm
T1183  ; M44->M45Auto RunOver Tm
T1200  ; 19.Axis Busy OffTm
T1201  ; 20.Axis Busy OffTm
T1202  ; 27.Axis Busy OffTm
T1203  ; 28.Axis Busy OffTm
T1221  ; L-BendInSideMoldPin Rev Tm
T1222  ; L-BendInSideMoldPinClampTm
T1223  ; L-BendInSideMoldPinUncmpTm
D11  ; L-BendOtMoldChanBuffer
D12  ; U-BendInMoldChanBuffer
D13  ; U-BendOtMoldChanBuffer
D16  ; Press   Working Set DataBuffer
D17  ; Buffer
D61  ; L,R     Select  Z-Bender
D300  ; Divert#1Model   Name Dis
D460  ; 31.Axis Set Data
D462  ; 32.Axis Set Data
D468  ; 150Ton  BackPushRev Pos'
D500  ; 1.Axis  Address Ok Range
D580  ; S/F Car'"A" Pos'Display &Set
D1100  ; L-BendInMoldMove#1 Data
D1104  ; L-BendInMoldMove#2 Data
D1106  ; L-BendInNow MoldData
D1110  ; L-BendOtMoldMove#1 Data
D1114  ; L-BendOtMoldMove#2 Data
D1116  ; L-BendOtNow MoldData
D1120  ; U-BendInMoldMove#1 Data
D1124  ; U-BendInMoldMove#2 Data
D1126  ; U-BendInNow MoldData
D1130  ; U-BendOtMoldMove#1 Data
D1134  ; U-BendOtMoldMove#2 Data
D1136  ; U-BendOtNow MoldData
D1210  ; Sheet#1 Total   Qty
D1300  ; CABINET SELECTION FROM BUFFER
D2030  ; Command PositionAxis-16
D2102  ; Auto    Speed   Set DataAxis-02
D2106  ; Auto    Speed   Set DataAxis-04
D2108  ; Auto    Speed   Set DataAxis-05
D2110  ; Auto    Speed   Set DataAxis-06
D2112  ; Auto    Speed   Set DataAxis-07
D2114  ; Auto    Speed   Set DataAxis-08
D2116  ; Auto    Speed   Set DataAxis-09
D2118  ; Auto    Speed   Set DataAxis-10
D2120  ; Auto    Speed   Set DataAxis-11
D2122  ; Auto    Speed   Set DataAxis-12
D2124  ; Auto    Speed   Set DataAxis-13
D2126  ; Auto    Speed   Set DataAxis-14
D2128  ; Auto    Speed   Set DataAxis-15
D2130  ; Auto    Speed   Set DataAxis-16
D2132  ; Auto    Speed   Set DataAxis-17
D2134  ; Auto    Speed   Set DataAxis-18
D2136  ; Auto    Speed   Set DataAxis-19
D2138  ; Auto    Speed   Set DataAxis-20
D2140  ; Auto    Speed   Set DataAxis-21
D2142  ; Auto    Speed   Set DataAxis-22
D2144  ; Auto    Speed   Set DataAxis-23
D2146  ; Auto    Speed   Set DataAxis-24
D2148  ; Auto    Speed   Set DataAxis-25
D2150  ; Auto    Speed   Set DataAxis-26
D2152  ; Auto    Speed   Set DataAxis-27
D2154  ; Auto    Speed   Set DataAxis-28
D2156  ; Auto    Speed   Set DataAxis-29
D2158  ; Auto    Speed   Set DataAxis-30
D2160  ; 31.Axis SetSpeedMove
D2162  ; 32.Axis SetSpeedMove
D2204  ; All     Servo   Ready
D3160  ; Current PositionAxis-03
D3220  ; Current PositionAxis-06
D3280  ; Current PositionAxis-09
D3300  ; Current PositionAxis-10
D3320  ; Current PositionAxis-11
D3340  ; Current PositionAxis-12
D3380  ; Current PositionAxis-14
D3420  ; Current PositionAxis-16
D3440  ; Current PositionAxis-17
D3460  ; Current PositionAxis-18
D3480  ; Current PositionAxis-19
D3520  ; Current PositionAxis-21
D3720  ; Current PositionAxis-31
D3740  ; Current PositionAxis-32
D4000  ; 1.Axis  Set DataMove
D4002  ; 2.Axis  Set DataMove
D4004  ; 3.Axis  Set DataMove
D4006  ; 4.Axis  Set DataMove
D4008  ; 5.Axis  Set DataMove
D4010  ; 6.Axis  Set DataMove
D4012  ; 7.Axis  Set DataMove
D4014  ; 8.Axis  Set DataMove
D4016  ; 9.Axis  Set DataMove
D4018  ; 10.Axis Set DataMove
D4020  ; 11.Axis Set DataMove
D4022  ; 12.Axis Set DataMove
D4024  ; 13.Axis Set DataMove
D4026  ; 14.Axis Set DataMove
D4028  ; 15.Axis Set DataMove
D4100  ; 1.Axis  Auto    Speed
D4102  ; 2.Axis  Auto    Speed
D4104  ; 3.Axis  Auto    Speed
D4106  ; 4.Axis  Auto    Speed
D4108  ; 5.Axis  Auto    Speed
D4110  ; 6.Axis  Auto    Speed
D4112  ; 7.Axis  Auto    Speed
D4114  ; 8.Axis  Auto    Speed
D4116  ; 9.Axis  Auto    Speed
D4118  ; 10.Axis Auto    Speed
D4120  ; 11.Axis Auto    Speed
D4122  ; 12.Axis Auto    Speed
D4124  ; 13.Axis Auto    Speed
D4126  ; 14.Axis Auto    Speed
D4128  ; 15.Axis Auto    Speed
W10  ; Tact    time  ofLQC     machine
W11  ; AVG     cycle   time
W12  ; Idel    time
W13  ; Idel    Time Feq
W14  ; Efficiency      Rate %
R11  ; Buffer  ModelNo.
R15  ; Taping#2ModelNo.
R50  ; 9.Axis  BackWaitSet Data
R52  ; JogSpeedFast
R60  ; 1.Axis  JogSpeedFast%
R62  ; 1.Axis  JogSpeedSlow%
R68  ; 9.Axis  JogSpeedFast%
R70  ; 9.Axis  JogSpeedSlow%
R100  ; L-BendInNow MoldData(EA)
R102  ; L-BenderMold 1EAPitchDat200mm
R104  ; L-BenderMoldMoveData400mm
R106  ; L-BendOtNow MoldData(EA)
R108  ; 19.Axis Set Data+
R110  ; L-BenderMold    Pitch   Data
R120  ; U-BendInNow MoldData(EA)
R122  ; U-BenderMold    Pitch   Data
R124  ; U-BenderMoldPitcNormal  Data
R126  ; U-BendOtNow MoldData(EA)
R128  ; 12.Axis Set Data-
R130  ; U-BenderMold    Pitch   Data
R250  ; Sheet#1 Main    SetCount
R260  ; Sheet#1 Main    Count
R261  ; Sheet#2 Main    Count
R262  ; Sheet#3 Main    Count
R263  ; Sheet#4 Main    Count
R264  ; Sheet#5 Main    Count
R265  ; S/F     Working Order 1
R280  ; Each    Model   PV Data
R291  ; S/F     Working Order 2
R292  ; S/F     Working Order 3
R293  ; S/F     Working Order 4
R294  ; S/F     Working Order 5
R295  ; S/F     Working Order 6
R296  ; S/F     Working Order 7
R297  ; S/F     Working Order 8
R402  ; MaxSpeedAxis-02
R404  ; MaxSpeedAxis-03
R406  ; MaxSpeedAxis-04
R408  ; MaxSpeedAxis-05
R410  ; MaxSpeedAxis-06
R412  ; MaxSpeedAxis-07
R414  ; MaxSpeedAxis-08
R416  ; MaxSpeedAxis-09
R418  ; MaxSpeedAxis-10
R420  ; MaxSpeedAxis-11
R426  ; MaxSpeedAxis-14
R430  ; MaxSpeedAxis-16
R434  ; MaxSpeedAxis-18
R446  ; MaxSpeedAxis-24
R448  ; MaxSpeedAxis-25
R450  ; MaxSpeedAxis-26
R458  ; MaxSpeedAxis-30
R502  ; Auto    Speed % Axis-02
R504  ; Auto    Speed % Axis-03
R506  ; Auto    Speed % Axis-04
R508  ; Auto    Speed % Axis-05
R510  ; Auto    Speed % Axis-06
R512  ; Auto    Speed % Axis-07
R514  ; Auto    Speed % Axis-08
R516  ; Auto    Speed % Axis-09
R518  ; Auto    Speed % Axis-10
R520  ; Auto    Speed % Axis-11
R522  ; Auto    Speed % Axis-12
R526  ; Auto    Speed % Axis-14
R528  ; Auto    Speed % Axis-15
R530  ; Auto    Speed % Axis-16
R532  ; Auto    Speed % Axis-17
R534  ; Auto    Speed % Axis-18
R538  ; Auto    Speed % Axis-20
R540  ; Auto    Speed % Axis-21
R542  ; Auto    Speed % Axis-22
R544  ; Auto    Speed % Axis-23
R546  ; Auto    Speed % Axis-24
R548  ; Auto    Speed % Axis-25
R550  ; Auto    Speed % Axis-26
R554  ; Auto    Speed % Axis-28
R556  ; Auto    Speed % Axis-29
R558  ; Auto    Speed % Axis-30
R560  ; 31.Axis Auto    Speed
R562  ; 32.Axis Auto    Speed
R602  ; +OT Set PositionAxis-02
R604  ; +OT Set PositionAxis-03
R606  ; +OT Set PositionAxis-04
R608  ; +OT Set PositionAxis-05
R610  ; +OT Set PositionAxis-06
R612  ; +OT Set PositionAxis-07
R614  ; +OT Set PositionAxis-08
R616  ; +OT Set PositionAxis-09
R618  ; +OT Set PositionAxis-10
R620  ; +OT Set PositionAxis-11
R622  ; +OT Set PositionAxis-12
R624  ; +OT Set PositionAxis-13
R626  ; +OT Set PositionAxis-14
R628  ; +OT Set PositionAxis-15
R630  ; +OT Set PositionAxis-16
R632  ; +OT Set PositionAxis-17
R634  ; +OT Set PositionAxis-18
R636  ; +OT Set PositionAxis-19
R638  ; +OT Set PositionAxis-20
R640  ; +OT Set PositionAxis-21
R642  ; +OT Set PositionAxis-22
R644  ; +OT Set PositionAxis-23
R646  ; +OT Set PositionAxis-24
R648  ; +OT Set PositionAxis-25
R650  ; +OT Set PositionAxis-26
R652  ; +OT Set PositionAxis-27
R654  ; +OT Set PositionAxis-28
R656  ; +OT Set PositionAxis-29
R658  ; +OT Set PositionAxis-30
R660  ; +OT Set PositionAxis-31
R662  ; +OT Set PositionAxis-32
R700  ; -OT Set PositionAxis-01
R702  ; -OT Set PositionAxis-02
R704  ; -OT Set PositionAxis-03
R706  ; -OT Set PositionAxis-04
R708  ; -OT Set PositionAxis-05
R710  ; -OT Set PositionAxis-06
R712  ; -OT Set PositionAxis-07
R714  ; -OT Set PositionAxis-08
R716  ; -OT Set PositionAxis-09
R718  ; -OT Set PositionAxis-10
R720  ; -OT Set PositionAxis-11
R722  ; -OT Set PositionAxis-12
R724  ; -OT Set PositionAxis-13
R726  ; -OT Set PositionAxis-14
R728  ; -OT Set PositionAxis-15
R730  ; -OT Set PositionAxis-16
R732  ; -OT Set PositionAxis-17
R734  ; -OT Set PositionAxis-18
R736  ; -OT Set PositionAxis-19
R738  ; -OT Set PositionAxis-20
R740  ; -OT Set PositionAxis-21
R742  ; -OT Set PositionAxis-22
R744  ; -OT Set PositionAxis-23
R746  ; -OT Set PositionAxis-24
R748  ; -OT Set PositionAxis-25
R750  ; -OT Set PositionAxis-26
R752  ; -OT Set PositionAxis-27
R754  ; -OT Set PositionAxis-28
R756  ; -OT Set PositionAxis-29
R758  ; -OT Set PositionAxis-30
R760  ; -OT Set PositionAxis-31
R762  ; -OT Set PositionAxis-32
R800  ; ModelNo1Name
R922  ; Set HomePos'DataAxis-12
R926  ; Set HomePos'DataAxis-14
R930  ; Set HomePos'DataAxis-16
R960  ; Set HomePos'DataAxis-31
R962  ; Set HomePos'DataAxis-32
R1000  ; 1.Axis  Set DataNo.A
R1002  ; 1.Axis  Set DataNo.B
R1004  ; 1.Axis  Set DataNo.C
R1006  ; 1.Axis  Set DataNo.D
R1008  ; 1.Axis  Set DataNo.E
R1010  ; 1.Axis  Set DataNo.F
R1012  ; 1.Axis  Set DataConv'
R1100  ; 2.Axis  Set DataNo.1
R1200  ; 3.Axis  Set DataNo.1
R1300  ; 4.Axis  Set DataNo.1
R1400  ; 5.Axis  Set DataNo.1
R1500  ; 6.Axis  Set DataNo.1
R1600  ; 7.Axis  Set DataNo.1
R1700  ; 8.Axis  Set DataNo.1
R1800  ; 9.Axis  Set DataNo.1
R1900  ; 10.Axis Set DataNo.1
R2000  ; 11.Axis Set DataNo.1
R2100  ; 12.Axis Set DataNo.1
R2200  ; 13.Axis Set Data
R2300  ; 14.Axis Set DataNo.1
R2400  ; 15.Axis Set DataNo.1
R2800  ; 19.Axis Set Data
R3000  ; 17.Axis Set DataNo.1
R3100  ; 18.Axis Set DataNo.1
R3200  ; 19.Axis Set DataNo.1
R3300  ; 20.Axis Set DataNo.1
R3400  ; 21.Axis Set DataNo.1
R3500  ; 22.Axis Set DataNo.1
R3600  ; 27.Axis Set Data
R3700  ; 24.Axis Set DataNo.1
R3800  ; 25.Axis Set DataNo.1
R3900  ; 26.Axis Set DataNo.1
R4000  ; 27.Axis Set DataNo.1
R4100  ; 28.Axis Set DataNo.1
R4200  ; Press   Working Set Data#1
R4300  ; Press   Working Set Data#2
R4400  ; 31.Axis Set DataNo.1
R5000  ; ModelNo1Name
R6000  ; S/F Jog High    Speed %
R6002  ; S/F Jog Slow    Speed %
R6004  ; S/F Jog High    Speed
R6012  ; S/F Jog Slow    Speed
R6020  ; Noching Wide JogHigh    Speed %
R6022  ; Noching Wide JogSlow    Speed %
R6024  ; Noching Wide JogHigh    Speed
R6026  ; Noching Wide JogHigh    Speed
R6028  ; Noching Wide JogSlow    Speed
R6032  ; Noching Head JogHigh    Speed
R6036  ; Noching Head JogSlow    Speed
R6040  ; 150 Ton Jog HighSpeed %
R6042  ; 150 Ton Jog SlowHigh    Speed %
R6044  ; 150 Ton Jog HighSpeed
R6046  ; 150 Ton Jog HighSpeed
R6050  ; 150 Ton Jog SlowHigh    Speed
R6052  ; 150 Ton Jog SlowHigh    Speed
R6060  ; RollFormJog HighSpeed %
R6062  ; RollFormJog SlowSpeed %
R6064  ; RollFormJog HighSpeed
R6066  ; RollFormJog HighSpeed
R6080  ; L-BenderJog HighSpeed %
R6082  ; L-BenderJog SlowSpeed %
R6084  ; L-BenderJog HighSpeed
R6088  ; L-BenderJog SlowSpeed
R6100  ; U-BenderJog HighSpeed %
R6102  ; U-BenderJog SlowSpeed %
R6104  ; 25.Axis High    Speed
R6108  ; 25.Axis Slow    Speed
R6120  ; 26.Axis Jog HighSpeed
R6124  ; 26.Axis Jog SlowSpeed
R6130  ; 27.28.  Axis JogHigh    Speed
R6134  ; 27.28.  Axis JogSlow    Speed
R6140  ; 29.Axis Jog HighSpeed
R6144  ; U-BenderJog SlowSpeed
R6150  ; 30.Axis Jog HighSpeed
R6154  ; 30.Axis Jog SlowSpeed
R6180  ; 19.20   Axis JogHigh    Speed
R6184  ; 19.20   Axis JogSlow    Speed
R6190  ; 21.22   Axis JogHigh    Speed
R6194  ; 21.22   Axis JogSlow    Speed
R22200  ; 13.Axis Set DataNo.1
